SUBAPPLICATION Start_Baumsetzer (* Subapplication Type *)
  (* Standard: 61499-2 *)
  (* Version 1.0, 2024-07-12, Elias *)
  PACKAGE FBs::Baumsetzer::func::Automatik;
  IMPORT NVS_Keys::Key_Summer_Reset_Store;
  IMPORT isobus::UT::io::Button::ButtonActivationCode::BT_RELEASED_UNLATCHED;
  IMPORT isobus::UT::io::Softkey::SoftKeyActivationCode::SK_RELEASED;
  IMPORT test::FBs::Baumsetzer::Constants::DefaultPool::Button_Reset_Einsatzdauer;
  IMPORT test::FBs::Baumsetzer::Constants::DefaultPool::Start;
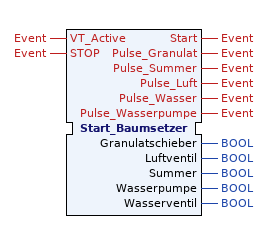
  EVENT_INPUT
    VT_Active;
    STOP; (* Stop Event *)
  END_EVENT
  EVENT_OUTPUT
    Start;
    Pulse_Granulat; (* Pulse *)
    Pulse_Summer;
    Pulse_Luft;
    Pulse_Wasser;
    Pulse_Wasserpumpe;
  END_EVENT
  VAR_OUTPUT
    Granulatschieber : BOOL; (* Granulatschieber *)
    Luftventil : BOOL; (* Luftventil *)
    Summer : BOOL; (* Summer *)
    Wasserpumpe : BOOL; (* Wasserpumpe *)
    Wasserventil : BOOL; (* Wasserventil *)
  END_VAR
  FBS
    E_CYCLE : iec61499::events::E_CYCLE(DT := T#1s);
    SoftKey_F1 : isobus::UT::io::Softkey::Softkey_IE(QI := TRUE, u16ObjId := Start, InputEvent := SK_RELEASED);
    SR_Wasserpumpe : iec61499::events::E_SR;
    Button_Reset_Einsatzdauer : isobus::UT::io::Button::Button_IE(QI := TRUE, u16ObjId := Button_Reset_Einsatzdauer, InputEvent := BT_RELEASED_UNLATCHED);
    GEN_PULSE_DIST : eclipse4diac::signalprocessing::distance::RangeBasedPulse(DIST_OFF := 0);
    GEN_PULSE_DIST_1 : eclipse4diac::signalprocessing::distance::RangeBasedPulse;
    GEN_PULSE_DIST_2 : eclipse4diac::signalprocessing::distance::RangeBasedPulse;
    GEN_PULSE_DIST_3 : eclipse4diac::signalprocessing::distance::RangeBasedPulse;
    E_PERMIT : iec61499::events::E_PERMIT;
    E_PERMIT_1 : iec61499::events::E_PERMIT;
    E_PERMIT_2 : iec61499::events::E_PERMIT;
    E_PERMIT_3 : iec61499::events::E_PERMIT;
    E_DELAY : iec61499::events::E_DELAY;
    E_SR : iec61499::events::E_SR;
    E_SR_1 : iec61499::events::E_SR;
    E_DELAY_1 : iec61499::events::E_DELAY;
    E_SR_2 : iec61499::events::E_SR;
    E_DELAY_2 : iec61499::events::E_DELAY;
    E_SR_3 : iec61499::events::E_SR;
    E_DELAY_3 : iec61499::events::E_DELAY;
    E_R_TRIG : iec61499::events::E_R_TRIG;
    E_R_TRIG_1 : iec61499::events::E_R_TRIG;
    E_R_TRIG_2 : iec61499::events::E_R_TRIG;
    E_R_TRIG_3 : iec61499::events::E_R_TRIG;
    E_F_TRIG : iec61499::events::E_F_TRIG;
    E_F_TRIG_1 : iec61499::events::E_F_TRIG;
    E_F_TRIG_2 : iec61499::events::E_F_TRIG;
    E_F_TRIG_3 : iec61499::events::E_F_TRIG;
    F_GT : iec61131::comparison::F_GT(IN2 := UDINT#0);
    E_CTU : iec61499::events::E_CTU;
    ADD_2 : iec61131::arithmetic::ADD_2;
    F_SUB : iec61131::arithmetic::F_SUB;
    NVS : logiBUS::storage::esp32_nvs::NVS(QI := TRUE, KEY := Key_Summer_Reset_Store, DEFAULT_VALUE := UDINT#0);
    E_PERMIT_6 : iec61499::events::E_PERMIT;
    F_MOVE : iec61131::selection::F_MOVE; {SET_ATTRIBUTE(DataType, UDINT)}
    F_MOVE_1 : iec61131::selection::F_MOVE; {SET_ATTRIBUTE(DataType, INT)}
    F_MOVE_2 : iec61131::selection::F_MOVE; {SET_ATTRIBUTE(DataType, INT)}
    F_EQ_DIRECTION : iec61131::comparison::F_EQ(IN2 := UDINT#1);
    E_PERMIT_5 : iec61499::events::E_PERMIT(PERMIT := TRUE);
    E_PERMIT_4 : iec61499::events::E_PERMIT;
    I_RHS : isobus::tecu::I_RHS(QI := TRUE);
    F_EQ_WORK_INDICATION : iec61131::comparison::F_EQ(IN2 := BYTE#1);
  END_FBS
  SUBAPPS
    Einsatzdauerzaehler : FBs::SlurryTanker::func::Zaehlermenue::Einsatzdauerzaehler;
    Einstellungen : FBs::Baumsetzer::func::Einstellungen::Einstellungen;
    Speed_Selection : FBs::Baumsetzer::func::Automatik::Speed_Selection;
  END_SUBAPPS
  EVENT_CONNECTIONS
    STOP TO SR_Wasserpumpe.R;
    SoftKey_F1.IND TO SR_Wasserpumpe.S;
    STOP TO E_CYCLE.STOP;
    SoftKey_F1.IND TO Start;
    E_CYCLE.EO TO Einsatzdauerzaehler.CountUp;
    Button_Reset_Einsatzdauer.IND TO Einsatzdauerzaehler.Reset;
    VT_Active TO Einsatzdauerzaehler.VT_Active;
    E_PERMIT.EO TO E_DELAY.START;
    E_PERMIT.EO TO E_SR.S;
    E_DELAY.EO TO E_SR.R;
    E_DELAY_1.EO TO E_SR_1.R;
    E_DELAY_2.EO TO E_SR_2.R;
    E_DELAY_3.EO TO E_SR_3.R;
    E_PERMIT_1.EO TO E_DELAY_1.START;
    E_PERMIT_1.EO TO E_SR_1.S;
    E_PERMIT_3.EO TO E_DELAY_3.START;
    E_PERMIT_3.EO TO E_SR_3.S;
    E_PERMIT_2.EO TO E_SR_2.S;
    E_PERMIT_2.EO TO E_DELAY_2.START;
    E_SR_1.EO TO Pulse_Summer;
    E_SR.EO TO Pulse_Granulat;
    E_SR_2.EO TO Pulse_Luft;
    E_SR_3.EO TO Pulse_Wasser;
    SR_Wasserpumpe.EO TO Pulse_Wasserpumpe;
    GEN_PULSE_DIST.CNF TO E_R_TRIG.EI;
    GEN_PULSE_DIST_1.CNF TO E_R_TRIG_1.EI;
    GEN_PULSE_DIST_3.CNF TO E_R_TRIG_3.EI;
    GEN_PULSE_DIST_2.CNF TO E_R_TRIG_2.EI;
    GEN_PULSE_DIST_2.CNF TO E_F_TRIG.EI;
    E_R_TRIG_2.EO TO E_PERMIT_2.EI;
    E_F_TRIG.EO TO E_PERMIT_2.EI;
    E_R_TRIG_1.EO TO E_PERMIT_1.EI;
    GEN_PULSE_DIST_1.CNF TO E_F_TRIG_1.EI;
    GEN_PULSE_DIST.CNF TO E_F_TRIG_2.EI;
    E_R_TRIG.EO TO E_PERMIT.EI;
    E_F_TRIG_2.EO TO E_PERMIT.EI;
    E_F_TRIG_1.EO TO E_PERMIT_1.EI;
    E_R_TRIG_3.EO TO E_PERMIT_3.EI;
    GEN_PULSE_DIST_3.CNF TO E_F_TRIG_3.EI;
    E_F_TRIG_3.EO TO E_PERMIT_3.EI;
    VT_Active TO E_CYCLE.START;
    SoftKey_F1.IND TO E_CTU.CU;
    STOP TO E_CTU.R;
    E_CTU.CUO TO F_GT.REQ;
    E_CTU.RO TO F_GT.REQ;
    F_GT.CNF TO E_PERMIT_6.EI;
    E_PERMIT_6.EO TO NVS.SET;
    NVS.SETO TO F_MOVE_1.REQ;
    NVS.GETO TO F_MOVE_1.REQ;
    F_MOVE_1.CNF TO F_SUB.REQ;
    F_SUB.CNF TO F_MOVE_2.REQ;
    F_MOVE_2.CNF TO ADD_2.REQ;
    E_PERMIT_5.EO TO F_MOVE.REQ;
    F_MOVE.CNF TO GEN_PULSE_DIST.REQ;
    F_MOVE.CNF TO GEN_PULSE_DIST_1.REQ;
    F_MOVE.CNF TO GEN_PULSE_DIST_2.REQ;
    F_MOVE.CNF TO GEN_PULSE_DIST_3.REQ;
    Speed_Selection.CNF TO F_EQ_DIRECTION.REQ;
    F_EQ_DIRECTION.CNF TO E_PERMIT_4.EI;
    E_PERMIT_4.EO TO E_PERMIT_5.EI;
    I_RHS.IND TO F_EQ_WORK_INDICATION.REQ;
    F_MOVE.CNF TO NVS.GET;
    Speed_Selection.CNF TO F_SUB.REQ;
  END_CONNECTIONS
  DATA_CONNECTIONS
    SR_Wasserpumpe.Q TO Wasserpumpe;
    Einstellungen.GranulatVersatz TO GEN_PULSE_DIST_1.DIST_OFF;
    Einstellungen.SummerDauer TO E_DELAY_1.DT;
    Einstellungen.GranulatDauer TO E_DELAY.DT;
    E_SR.Q TO Granulatschieber;
    E_SR_1.Q TO Summer;
    E_SR_2.Q TO Luftventil;
    E_SR_3.Q TO Wasserventil;
    Einstellungen.LuftDauer TO E_DELAY_2.DT;
    Einstellungen.WasserDauer TO E_DELAY_3.DT;
    GEN_PULSE_DIST.Q TO E_R_TRIG.QI;
    GEN_PULSE_DIST_1.Q TO E_R_TRIG_1.QI;
    GEN_PULSE_DIST_3.Q TO E_R_TRIG_3.QI;
    GEN_PULSE_DIST_2.Q TO E_R_TRIG_2.QI;
    Einstellungen.PflanzenAbstand TO GEN_PULSE_DIST_1.DIST_LOW;
    Einstellungen.PflanzenAbstand TO GEN_PULSE_DIST.DIST_LOW;
    Einstellungen.PflanzenAbstand TO GEN_PULSE_DIST_2.DIST_LOW;
    Einstellungen.PflanzenAbstand TO GEN_PULSE_DIST_3.DIST_LOW;
    Einstellungen.PflanzenAbstand TO GEN_PULSE_DIST_2.DIST_HIGH;
    Einstellungen.PflanzenAbstand TO GEN_PULSE_DIST.DIST_HIGH;
    Einstellungen.PflanzenAbstand TO GEN_PULSE_DIST_1.DIST_HIGH;
    Einstellungen.PflanzenAbstand TO GEN_PULSE_DIST_3.DIST_HIGH;
    GEN_PULSE_DIST_2.Q TO E_F_TRIG.QI;
    SR_Wasserpumpe.Q TO E_PERMIT_2.PERMIT;
    GEN_PULSE_DIST_1.Q TO E_F_TRIG_1.QI;
    GEN_PULSE_DIST.Q TO E_F_TRIG_2.QI;
    SR_Wasserpumpe.Q TO E_PERMIT.PERMIT;
    SR_Wasserpumpe.Q TO E_PERMIT_1.PERMIT;
    GEN_PULSE_DIST_3.Q TO E_F_TRIG_3.QI;
    SR_Wasserpumpe.Q TO E_PERMIT_3.PERMIT;
    Einstellungen.LuftVersatz TO GEN_PULSE_DIST_2.DIST_OFF;
    Einstellungen.WasserVersatz TO GEN_PULSE_DIST_3.DIST_OFF;
    E_CTU.CV TO F_GT.IN1;
    F_GT.OUT TO E_PERMIT_6.PERMIT;
    Einstellungen.PflanzenAbstand TO ADD_2.IN2;
    Speed_Selection.Distance TO F_SUB.IN1;
    Speed_Selection.Distance TO NVS.VALUE;
    NVS.VALUEO TO F_MOVE_1.IN;
    F_MOVE_1.OUT TO F_SUB.IN2;
    F_SUB.OUT TO F_MOVE_2.IN;
    F_MOVE_2.OUT TO ADD_2.IN1;
    ADD_2.OUT TO F_MOVE.IN;
    F_MOVE.OUT TO GEN_PULSE_DIST.DIST_IN;
    F_MOVE.OUT TO GEN_PULSE_DIST_1.DIST_IN;
    F_MOVE.OUT TO GEN_PULSE_DIST_2.DIST_IN;
    F_MOVE.OUT TO GEN_PULSE_DIST_3.DIST_IN;
    Speed_Selection.Direction TO F_EQ_DIRECTION.IN1;
    F_EQ_DIRECTION.OUT TO E_PERMIT_4.PERMIT;
    I_RHS.REAR_HITCH_WORK_INDICATION TO F_EQ_WORK_INDICATION.IN1;
  END_CONNECTIONS
END_SUBAPPLICATION
